TYPE T_CodePIT : STRING[7];
END_TYPE

(* stored: Version 1.1.0.1
   DUT T_CodePIT: Id {0148b596-6c5e-4926-8373-25ccd9a71555} *)
